{attribute 'linkalways'} 
{attribute 'no_explicit_call' := 'This FB is a CLASS and must be accessed using methods or properties'}
{attribute 'enable_dynamic_creation'}
FUNCTION_BLOCK AddAxisToGroupCommand EXTENDS NciCommand
VAR
	_fb : CfgAddAxisToGroup;
	_groupId : UDINT;
	_axisId : UDINT;
	_index : UDINT;
	_timeout : TIME;
END_VAR

METHOD FB_init : BOOL
VAR_INPUT
	bInitRetains : BOOL; // if TRUE, the retain variables are initialized (warm start / cold start)
	bInCopyCode : BOOL;  // if TRUE, the instance afterwards gets moved into the copy code (online change)
	nci : I_Nci;
	axis : I_Axis;
	index : UDINT;
	timeout : TIME;
END_VAR
IF nci <> 0 THEN
	_groupId := nci.GroupId;
END_IF
IF axis <> 0 THEN
	_axisId := axis.AxisId;
END_IF
_index := index;
_timeout := timeout;
END_METHOD

METHOD PROTECTED  WhileBusy
VAR_INPUT
	CommandState : I_CommandBusyState;
END_VAR
_fb(
	bExecute := TRUE,
	nGroupId := _groupId,
	nAxisId := _axisId,
	nIndex := _index,
	tTimeOut := _timeout
);

IF _fb.bBusy THEN
	RETURN;
END_IF

IF _fb.bErr THEN
	_fb(bExecute := FALSE);
	CommandState.SetError(_fb.nErrId);
	RETURN;
END_IF

_fb(bExecute := FALSE);
CommandState.SetDone();
END_METHOD

END_FUNCTION_BLOCK

(* stored: Version 1.1.0.1, ProductVersion 3.1.4024.12
   POU AddAxisToGroupCommand: Id {b565b1a5-a20d-0448-04e3-a1d11ba34f8a}, SpecialFunc None
   Method FB_init: Id {0145e603-67db-0365-11ad-f02d67fef8e9}
   Method WhileBusy: Id {a2a35993-d914-0900-38f3-f49e75bed586} *)
